// TIA Portal V17 export
// export: Created 2025-01-20T09:49:20.3609272Z, ExportSetting WithDefaults, DisplayName Totally Integrated Automation Portal, DisplayVersion V17 Update 7, DisplayName TIA Portal Openness, DisplayVersion V17 Update 7, DisplayName TIA Portal Version Control Interface, DisplayVersion V17, DisplayName SINAMICS Startdrive Advanced, DisplayVersion V17 SP2, DisplayName SINAMICS Startdrive G110M, G120, G120C, G120D, G120P, G115D, DisplayVersion V17 SP2, DisplayName SINAMICS Startdrive G130, G150, S120, S150, SINAMICS MV, S210, DisplayVersion V17 SP2, DisplayName STEP 7 Professional, DisplayVersion V17 Update 7, DisplayName STEP 7 Safety, DisplayVersion V17 Update 6, DisplayName WinCC Professional, DisplayVersion V17 Update 7
DATA_BLOCK "Block_2_DB"   // DB1
VERSION : 0.1
// stored: AutoNumber true, InstanceOfName Block_2, InstanceOfType FB
"Block_2"
   // VAR_INPUT
   //    "1" : Bool;
   // END_VAR
   // VAR_OUTPUT
   //    "2" : Bool;
   // END_VAR
BEGIN
END_DATA_BLOCK
